FUNCTION_BLOCK SludgeHoldingTank (* CAT Function Block Type *)
  (* Standard: 61499-2 *)
  (* Version 0.0, 27/08/2026, Schneider Electric, template *)
  PACKAGE Main;
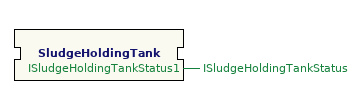
  PLUGS
    ISludgeHoldingTankStatus1 : ISludgeHoldingTankStatus;
  END_PLUGS
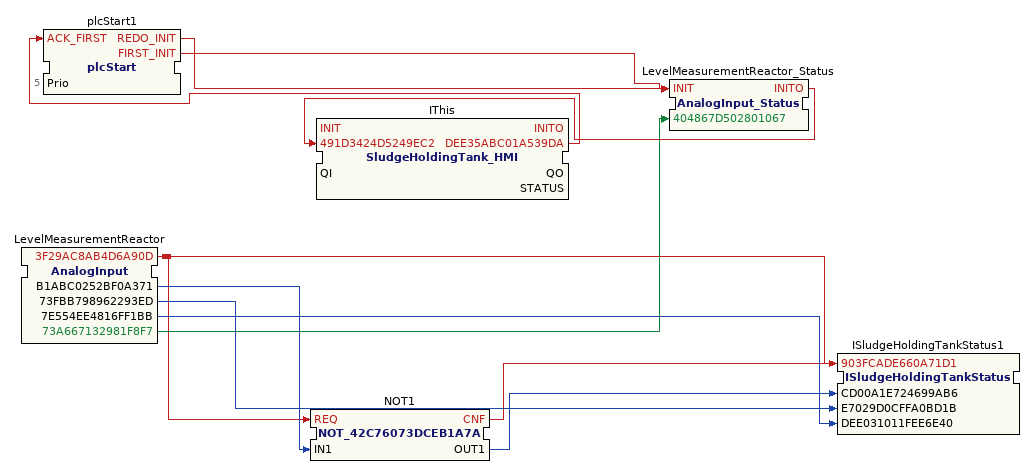
  FBS
    LevelMeasurementReactor_Status : AnalogInput_Status;
    LevelMeasurementReactor : AnalogInput;
    NOT1 : NOT_42C76073DCEB1A7A; {SET_ATTRIBUTE(Configuration.GenericFBType.InterfaceParams, Runtime.Standard#CNT:=1;OUT${CNT$}:BOOL)}
    plcStart1 : plcStart(Prio := 5);
    IThis : SludgeHoldingTank_HMI;
  END_FBS
  EVENT_CONNECTIONS
    LevelMeasurementReactor.3F29AC8AB4D6A90D TO NOT1.REQ;
    NOT1.CNF TO ISludgeHoldingTankStatus1.903FCADE660A71D1;
    plcStart1.REDO_INIT TO LevelMeasurementReactor_Status.INIT;
    plcStart1.FIRST_INIT TO LevelMeasurementReactor_Status.INIT;
    LevelMeasurementReactor_Status.INITO TO IThis.491D3424D5249EC2;
    IThis.DEE35ABC01A539DA TO plcStart1.ACK_FIRST;
    LevelMeasurementReactor.3F29AC8AB4D6A90D TO ISludgeHoldingTankStatus1.903FCADE660A71D1;
  END_CONNECTIONS
  DATA_CONNECTIONS
    LevelMeasurementReactor.B1ABC0252BF0A371 TO NOT1.IN1;
    NOT1.OUT1 TO ISludgeHoldingTankStatus1.CD00A1E724699AB6;
    LevelMeasurementReactor.73FBB798962293ED TO ISludgeHoldingTankStatus1.E7029D0CFFA0BD1B;
    LevelMeasurementReactor.7E554EE4816FF1BB TO ISludgeHoldingTankStatus1.DEE031011FEE6E40;
  END_CONNECTIONS
  ADAPTER_CONNECTIONS
    LevelMeasurementReactor.73A667132981F8F7 TO LevelMeasurementReactor_Status.404867D502801067;
  END_CONNECTIONS
END_FUNCTION_BLOCK
